# EPICS substitutions: iocBoot/ioc13bmd_DAC_XPS/XPSAux.substitutions
file "$(MOTOR)/db/XPSAuxLi.db"
{
pattern
{P,     R,          PORT,       CHAN,   SCAN}
{13BMD:,  XPSAux1Li,  XPS_AUX1,   0,      "I/O Intr"}
{13BMD:,  XPSAux2Li,  XPS_AUX1,   1,      "I/O Intr"}
{13BMD:,  XPSAux3Li,  XPS_AUX1,   2,      "I/O Intr"}
{13BMD:,  XPSAux4Li,  XPS_AUX1,   3,      "I/O Intr"}
}

file "$(MOTOR)/db/XPSAuxBi.db"
{
pattern
{P,    R,           PORT,     CHAN,  MASK,     SCAN}
{13BMD:, XPSAux1Bi0,  XPS_AUX1, 0,     0x000001, "I/O Intr"}
{13BMD:, XPSAux1Bi1,  XPS_AUX1, 0,     0x000002, "I/O Intr"}
{13BMD:, XPSAux1Bi2,  XPS_AUX1, 0,     0x000004, "I/O Intr"}
{13BMD:, XPSAux1Bi3,  XPS_AUX1, 0,     0x000008, "I/O Intr"}
{13BMD:, XPSAux1Bi4,  XPS_AUX1, 0,     0x000010, "I/O Intr"}
{13BMD:, XPSAux1Bi5,  XPS_AUX1, 0,     0x000020, "I/O Intr"}
{13BMD:, XPSAux1Bi6,  XPS_AUX1, 0,     0x000040, "I/O Intr"}
{13BMD:, XPSAux1Bi7,  XPS_AUX1, 0,     0x000080, "I/O Intr"}
{13BMD:, XPSAux2Bi0,  XPS_AUX1, 1,     0x000001, "I/O Intr"}
{13BMD:, XPSAux2Bi1,  XPS_AUX1, 1,     0x000002, "I/O Intr"}
{13BMD:, XPSAux2Bi2,  XPS_AUX1, 1,     0x000004, "I/O Intr"}
{13BMD:, XPSAux2Bi3,  XPS_AUX1, 1,     0x000008, "I/O Intr"}
{13BMD:, XPSAux2Bi4,  XPS_AUX1, 1,     0x000010, "I/O Intr"}
{13BMD:, XPSAux2Bi5,  XPS_AUX1, 1,     0x000020, "I/O Intr"}
{13BMD:, XPSAux3Bi0,  XPS_AUX1, 2,     0x000001, "I/O Intr"}
{13BMD:, XPSAux3Bi1,  XPS_AUX1, 2,     0x000002, "I/O Intr"}
{13BMD:, XPSAux3Bi2,  XPS_AUX1, 2,     0x000004, "I/O Intr"}
{13BMD:, XPSAux3Bi3,  XPS_AUX1, 2,     0x000008, "I/O Intr"}
{13BMD:, XPSAux3Bi4,  XPS_AUX1, 2,     0x000010, "I/O Intr"}
{13BMD:, XPSAux3Bi5,  XPS_AUX1, 2,     0x000020, "I/O Intr"}
{13BMD:, XPSAux4Bi0,  XPS_AUX1, 3,     0x000001, "I/O Intr"}
{13BMD:, XPSAux4Bi1,  XPS_AUX1, 3,     0x000002, "I/O Intr"}
{13BMD:, XPSAux4Bi2,  XPS_AUX1, 3,     0x000004, "I/O Intr"}
{13BMD:, XPSAux4Bi3,  XPS_AUX1, 3,     0x000008, "I/O Intr"}
{13BMD:, XPSAux4Bi4,  XPS_AUX1, 3,     0x000010, "I/O Intr"}
{13BMD:, XPSAux4Bi5,  XPS_AUX1, 3,     0x000020, "I/O Intr"}
{13BMD:, XPSAux4Bi6,  XPS_AUX1, 3,     0x000040, "I/O Intr"}
{13BMD:, XPSAux4Bi7,  XPS_AUX1, 3,     0x000080, "I/O Intr"}
{13BMD:, XPSAux4Bi8,  XPS_AUX1, 3,     0x000100, "I/O Intr"}
{13BMD:, XPSAux4Bi9,  XPS_AUX1, 3,     0x000200, "I/O Intr"}
{13BMD:, XPSAux4Bi10, XPS_AUX1, 3,     0x000400, "I/O Intr"}
{13BMD:, XPSAux4Bi11, XPS_AUX1, 3,     0x000800, "I/O Intr"}
{13BMD:, XPSAux4Bi12, XPS_AUX1, 3,     0x001000, "I/O Intr"}
{13BMD:, XPSAux4Bi13, XPS_AUX1, 3,     0x002000, "I/O Intr"}
{13BMD:, XPSAux4Bi14, XPS_AUX1, 3,     0x004000, "I/O Intr"}
{13BMD:, XPSAux4Bi15, XPS_AUX1, 3,     0x008000, "I/O Intr"}
}

file "$(MOTOR)/db/XPSAuxBo.db"
{
pattern
{P,    R,           PORT,     CHAN, MASK}
{13BMD:, XPSAux1Bo0,  XPS_AUX1, 0,    0x000001}
{13BMD:, XPSAux1Bo1,  XPS_AUX1, 0,    0x000002}
{13BMD:, XPSAux1Bo2,  XPS_AUX1, 0,    0x000004}
{13BMD:, XPSAux1Bo3,  XPS_AUX1, 0,    0x000008}
{13BMD:, XPSAux1Bo4,  XPS_AUX1, 0,    0x000010}
{13BMD:, XPSAux1Bo5,  XPS_AUX1, 0,    0x000020}
{13BMD:, XPSAux1Bo6,  XPS_AUX1, 0,    0x000040}
{13BMD:, XPSAux1Bo7,  XPS_AUX1, 0,    0x000080}
{13BMD:, XPSAux3Bo0,  XPS_AUX1, 1,    0x000001}
{13BMD:, XPSAux3Bo1,  XPS_AUX1, 1,    0x000002}
{13BMD:, XPSAux3Bo2,  XPS_AUX1, 1,    0x000004}
{13BMD:, XPSAux3Bo3,  XPS_AUX1, 1,    0x000008}
{13BMD:, XPSAux3Bo4,  XPS_AUX1, 1,    0x000010}
{13BMD:, XPSAux3Bo5,  XPS_AUX1, 1,    0x000020}
{13BMD:, XPSAux4Bo0,  XPS_AUX1, 2,    0x000001}
{13BMD:, XPSAux4Bo1,  XPS_AUX1, 2,    0x000002}
{13BMD:, XPSAux4Bo2,  XPS_AUX1, 2,    0x000004}
{13BMD:, XPSAux4Bo3,  XPS_AUX1, 2,    0x000008}
{13BMD:, XPSAux4Bo4,  XPS_AUX1, 2,    0x000010}
{13BMD:, XPSAux4Bo5,  XPS_AUX1, 2,    0x000020}
{13BMD:, XPSAux4Bo6,  XPS_AUX1, 2,    0x000040}
{13BMD:, XPSAux4Bo7,  XPS_AUX1, 2,    0x000080}
{13BMD:, XPSAux4Bo8,  XPS_AUX1, 2,    0x000100}
{13BMD:, XPSAux4Bo9,  XPS_AUX1, 2,    0x000200}
{13BMD:, XPSAux4Bo10, XPS_AUX1, 2,    0x000400}
{13BMD:, XPSAux4Bo11, XPS_AUX1, 2,    0x000800}
{13BMD:, XPSAux4Bo12, XPS_AUX1, 2,    0x001000}
{13BMD:, XPSAux4Bo13, XPS_AUX1, 2,    0x002000}
{13BMD:, XPSAux4Bo14, XPS_AUX1, 2,    0x004000}
{13BMD:, XPSAux4Bo15, XPS_AUX1, 2,    0x008000}
}

file "$(MOTOR)/db/XPSAuxLo.db"
{
pattern
{P,     R,         PORT,     CHAN}
{13BMD:,  XPSAux1Lo, XPS_AUX1, 0}
{13BMD:,  XPSAux3Lo, XPS_AUX1, 1}
{13BMD:,  XPSAux4Lo, XPS_AUX1, 2}
}

file "$(MOTOR)/db/XPSAuxAi.db"
{
pattern
{P,    R,          PORT,     CHAN, LOPR,   HOPR,  PREC, SCAN}
{13BMD:, XPSAuxAi0,  XPS_AUX1, 0,    -10.0,  10.0,  4,    "1 second"}
{13BMD:, XPSAuxAi1,  XPS_AUX1, 1,    -10.0,  10.0,  4,    "1 second"}
{13BMD:, XPSAuxAi2,  XPS_AUX1, 2,    -10.0,  10.0,  4,    "1 second"}
{13BMD:, XPSAuxAi3,  XPS_AUX1, 3,    -10.0,  10.0,  4,    "1 second"}
}

file "$(MOTOR)/db/XPSAuxAo.db"
{
pattern
{P,    R,          PORT,     CHAN, DRVL,   LOPR,   DRVH,  HOPR,  PREC}
{13BMD:, XPSAuxAo0,  XPS_AUX1, 0,    -10.0,  -10.0,  10.0,  10.0,   4}
{13BMD:, XPSAuxAo1,  XPS_AUX1, 1,    -10.0,  -10.0,  10.0,  10.0,   4}
{13BMD:, XPSAuxAo2,  XPS_AUX1, 2,    -10.0,  -10.0,  10.0,  10.0,   4}
{13BMD:, XPSAuxAo3,  XPS_AUX1, 3,    -10.0,  -10.0,  10.0,  10.0    4}
}
